FUNCTION_BLOCK FB_Stepper EXTENDS FB_AxisNc
VAR_INPUT
	nStatusByte : BYTE;
END_VAR
VAR_OUTPUT
	nCtrlByte : BYTE; 
END_VAR
VAR
END_VAR

METHOD PUBLIC M_HardwareReset : UDINT
//Set bit 6 in the Control word that will be transmitted to the stepper for resetting. 
VAR_INPUT
	bReset : BOOL;
END_VAR
//REturn 0 when idle
//Return 1 when busy 
//return 3 when complete
VAR_INST // added by the converter: edge detectors and wires of the graphical bodies
    _w1, _w2 : BOOL;
    _w3, _w4 : ANY;
END_VAR
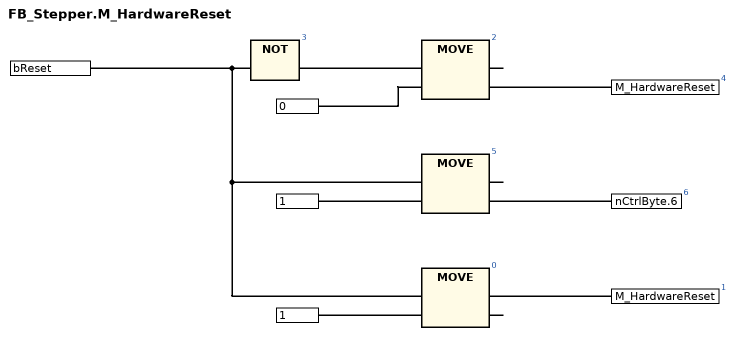
_w1 := bReset;
IF _w1 THEN (* 1; result not used *) END_IF
M_HardwareReset := _w1;
IF _w2 THEN _w3 := 0; END_IF
_w2 := NOT bReset;
M_HardwareReset := _w3;
IF bReset THEN _w4 := 1; END_IF
nCtrlByte.6 := _w4;
END_METHOD

END_FUNCTION_BLOCK

(* stored: Version 1.1.0.1, ProductVersion 3.1.4024.11
   POU FB_Stepper: Id {08ef0f76-aa6d-422b-a4bd-1a08ac9ff1fa}, SpecialFunc None
   Method M_HardwareReset: Id {b5f41d3d-f473-4f27-b358-0c1b3c43d744} *)
